FUNCTION_BLOCK AB_STOP (* Basic FB with empty ECC *)
  (* Standard: 61499-2 *)
  (* Version 1.0, 2023-01-19, Alex Maximov *)
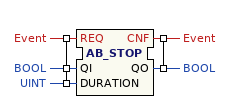
  EVENT_INPUT
    REQ WITH QI, DURATION;
  END_EVENT
  EVENT_OUTPUT
    CNF WITH QO;
  END_EVENT
  VAR_INPUT
    QI : BOOL;
    DURATION : UINT;
  END_VAR
  VAR_OUTPUT
    QO : BOOL;
  END_VAR
  EC_STATES
    START; (* Initial State *)
  END_STATES
END_FUNCTION_BLOCK
